# B&R Automation Studio project perfxxl (part 5)

#### motorman.c
```c
#ifdef _DEFAULT_INCLUDES
	#include <AsDefault.h>
#endif
/*
                             *******************
******************************* C SOURCE FILE *******************************
**                           *******************                           **
**                                                                         **
** project  : LS JET II                                                    **
** filename : MOTORMAN.C                                                   **
** version  : 1.11                                                         **
** date     : 08.11.2007                                                   **
**                                                                         **
*****************************************************************************
** Abstract                                                                **
** ========                                                                **
** Move motor manually                                                     **
**                                                                         **
**                                                                         **
** Copyright (c) 2006, Krause-Biagosch GmbH                                **
** All rights reserved.                                                    **
**                                                                         **
*****************************************************************************
VERSION HISTORY:
----------------
Version     : 1.00
Date        : 10.09.2002
Revised by  : Herbert Aden
Description : Original version.

Version     : 1.10
Date        : 07.11.2006
Revised by  : Herbert Aden
Description : -Code review, style improvement

Version     : 1.11
Date        : 08.11.2007
Revised by  : Herbert Aden
Description : - limits for checking movement are now always positive, and max>min
*/
#define _MOTORMAN_C_SRC

/****************************************************************************/
/**                                                                        **/
/**                           INCLUDE FILES                                **/
/**                                                                        **/
/****************************************************************************/
#include <string.h>
#include "asstring.h"
#include "glob_var.h"
#include "Motorfunc.h"

/****************************************************************************/
/**                                                                        **/
/**                       DEFINITIONS AND MACROS                           **/
/**                                                                        **/
/****************************************************************************/
/* NONE */

/****************************************************************************/
/**                                                                        **/
/**                      TYPEDEFS AND STRUCTURES                           **/
/**                                                                        **/
/****************************************************************************/
/* NONE */

/****************************************************************************/
/**                                                                        **/
/**                      PROTOTYPES OF LOCAL FUNCTIONS                     **/
/**                                                                        **/
/****************************************************************************/
/* NONE */

/****************************************************************************/
/**                                                                        **/
/**                      EXPORTED VARIABLES                                **/
/**                                                                        **/
/****************************************************************************/
/* NONE */

/****************************************************************************/
/**                                                                        **/
/**                           GLOBAL VARIABLES                             **/
/**                                                                        **/
/****************************************************************************/
_GLOBAL   UINT                ConveyorBeltOn;

/****************************************************************************/
/**                                                                        **/
/**                      TASK-LOCAL VARIABLES                              **/
/**                                                                        **/
/****************************************************************************/
_LOCAL    USINT               ManStep;
_LOCAL    USINT               MotorOnDisplay;
_LOCAL    USINT               ManPlus,ManMinus;

/****************************************************************************/
/**                                                                        **/
/**                    MODULE-LOCAL VARIABLES                              **/
/**                                                                        **/
/****************************************************************************/
static    DINT                tmpval;

/****************************************************************************/
/**                                                                        **/
/**                          EXPORTED FUNCTIONS                            **/
/**                                                                        **/
/****************************************************************************/
void MotorManual(void)
{
	MotorOnDisplay = gMotorOnDisplay;
	switch (ManStep)
	{
		case 0:
		{
			if(Motors[MotorOnDisplay].Error || MotorOnDisplay == 0)
				break;

/* don't start, if limit reached*/
			if ((MotorOnDisplay != CONVEYORBELT) && (MotorOnDisplay != ADJUSTER))
			{
				if( ( ManPlus &&
				      (labs(Motors[MotorOnDisplay].Position) > labs(Motors[MotorOnDisplay].Parameter.MaximumPosition))
				    )
				 ||
				    ( ManMinus &&
					 (labs(Motors[MotorOnDisplay].Position) < labs(Motors[MotorOnDisplay].Parameter.MinimumPosition))
				    )
				  )
				{
					break;
				}
			}

			if( ManPlus || ManMinus )
			{
				ManStep = 1;
				if( ManMinus )
					tmpval = (-1L) * labs(Motors[MotorOnDisplay].Parameter.ManSpeed);
				else
					tmpval = labs(Motors[MotorOnDisplay].Parameter.ManSpeed);
			}
			break;
		}
		case 1:
		{
			if (SendMotorCmd(MotorOnDisplay, CMD_SERIAL, FALSE, 0L ))
			{
				ManStep = 2;
			}
			break;
		}
		case 2:
		{
			if (SendMotorCmd(MotorOnDisplay, CMD_MOVE_AT, TRUE, tmpval ))
			{
				ManStep = 3;
			}
			break;
		}
		case 3:
		{
/*wait for key being released*/
/*V2.10 or limit reached*/
/*V2.13 build 22.06.2005 no limits for Motor 6 and 9 (Belt-motors)*/
			if ((MotorOnDisplay != CONVEYORBELT) && (MotorOnDisplay != ADJUSTER))
			{
				if( ( ManPlus &&
				      (labs(Motors[MotorOnDisplay].Position) > labs(Motors[MotorOnDisplay].Parameter.MaximumPosition))
				    )
				 ||
				    ( ManMinus &&
					 (labs(Motors[MotorOnDisplay].Position) < labs(Motors[MotorOnDisplay].Parameter.MinimumPosition))
				    )
				  )
				{
					ManStep = 4;
					break;
				}
			}

			if( ManPlus || ManMinus )
				break;
			else
				ManStep = 4;

			break;
		}
		case 4:
		{
			if (SendMotorCmd(MotorOnDisplay, CMD_STOP, FALSE, 0L) )
			{
				ManStep = 0;
				if(MotorOnDisplay == CONVEYORBELT)
					ConveyorBeltOn = FALSE;
			}
			break;
		}
	}
}
/****************************************************************************/
/**                                                                        **/
/**                                 EOF                                    **/
/**                                                                        **/
/****************************************************************************/
```

#### motortarget.c
```c
#ifdef _DEFAULT_INCLUDES
	#include <AsDefault.h>
#endif
/*
                             *******************
******************************* C SOURCE FILE *******************************
**                           *******************                           **
**                                                                         **
** project  : LS JET II                                                    **
** filename : MOTORTARGET.C                                                **
** version  : 1.11                                                         **
** date     : 12.10.2007                                                   **
**                                                                         **
*****************************************************************************
** Abstract                                                                **
** ========                                                                **
** Sequence for moving a motor to a certain position (manually)            **
**                                                                         **
**                                                                         **
** Copyright (c) 2006, Krause-Biagosch GmbH                                **
** All rights reserved.                                                    **
**                                                                         **
*****************************************************************************
VERSION HISTORY:
----------------
Version     : 1.00
Date        : 10.09.2002
Revised by  : Herbert Aden
Description : Original version.

Version     : 1.10
Date        : 07.11.2006
Revised by  : Herbert Aden
Description : -Code review, style improvement

Version     : 1.10
Date        : 12.10.2007
Revised by  : Herbert Aden
Description : MoveToAbsPosition has changed, so we must provide a pointer
              to an USINT variable that can hold the internal state of that fct.
*/
#define _MOTORTARGET_C_SRC

/****************************************************************************/
/**                                                                        **/
/**                           INCLUDE FILES                                **/
/**                                                                        **/
/****************************************************************************/
#include <string.h>
#include "asstring.h"
#include "glob_var.h"
#include "Motorfunc.h"

/****************************************************************************/
/**                                                                        **/
/**                       DEFINITIONS AND MACROS                           **/
/**                                                                        **/
/****************************************************************************/
/* NONE */

/****************************************************************************/
/**                                                                        **/
/**                      PROTOTYPES OF LOCAL FUNCTIONS                     **/
/**                                                                        **/
/****************************************************************************/
/* NONE */

/****************************************************************************/
/**                                                                        **/
/**                      EXPORTED VARIABLES                                **/
/**                                                                        **/
/****************************************************************************/
/* NONE */

/****************************************************************************/
/**                                                                        **/
/**                           GLOBAL VARIABLES                             **/
/**                                                                        **/
/****************************************************************************/
/* NONE */

/****************************************************************************/
/**                                                                        **/
/**                      TASK-LOCAL VARIABLES                              **/
/**                                                                        **/
/****************************************************************************/
_LOCAL USINT	TargetStep;
_LOCAL USINT	MotorOnDisplay;
_LOCAL USINT	TargetStart;
_LOCAL DINT	TargetPosition;

/****************************************************************************/
/**                                                                        **/
/**                    MODULE-LOCAL VARIABLES                              **/
/**                                                                        **/
/****************************************************************************/
static    USINT               MotStep;       /* holds current step of fct MoveToAbsPosition */

/****************************************************************************/
/**                                                                        **/
/**                          EXPORTED FUNCTIONS                            **/
/**                                                                        **/
/****************************************************************************/
void MotorTarget(void)
{
	switch (TargetStep)
	{
		case 0:
		{
			if(		(Motors[MotorOnDisplay].Error == TRUE)
			    ||  (Motors[MotorOnDisplay].ReferenceOk == FALSE)
				||	(MotorOnDisplay == 0) )
				break;

/*check limit positions*/
			if ((MotorOnDisplay != CONVEYORBELT) && (MotorOnDisplay != ADJUSTER))
			{
				if(		(labs(TargetPosition) > labs(Motors[MotorOnDisplay].Parameter.MaximumPosition) )
					||	(labs(TargetPosition) < labs(Motors[MotorOnDisplay].Parameter.MinimumPosition)) )
					break;
			}

			if( TargetStart)
			{
				TargetStep = 1;
				TargetStart = FALSE;
			}
			break;
		}
		case 1:
		{
/*wait, till no other sending active*/
			if( MoveToAbsPosition(MotorOnDisplay,
			                      TargetPosition,
			                      Motors[MotorOnDisplay].Parameter.ManSpeed,
			                      &MotStep) )
			{
				TargetStep = 4;
			}
			break;
		}
		case 4:
		{
/*set maximum speed*/
			if( SendMotorCmd(MotorOnDisplay,
			                 CMD_SPEED,
			                 TRUE,
			                 Motors[MotorOnDisplay].Parameter.MaximumSpeed) )
			{
				TargetStep = 0;
			}
			break;
		}
	}
/*always reset the start command unconditionally*/
	TargetStart = FALSE;

}
/****************************************************************************/
/**                                                                        **/
/**                                 EOF                                    **/
/**                                                                        **/
/****************************************************************************/
```

#### motorstop.c
```c
#ifdef _DEFAULT_INCLUDES
	#include <AsDefault.h>
#endif
/****************************************************************************/
/*	Stoppen aller Motoren (quasi NOTAUS)*/
/*																			*/
/*																			*/
/*	Versionsgeschichte:														*/
/*  Version		Datum		Änderung								von		*/
/*	1.0			30.06.03	erste Implementation					HA		*/
/*																			*/
/*																			*/
/****************************************************************************/
#include "glob_var.h"
#include "in_out.h"
#include "asstring.h"
#include <string.h>
#include "motorfunc.h"

#define BROADCAST 127

_LOCAL 	USINT	StopStep;
_LOCAL F_TRIGtyp F_DoorSensor;

_GLOBAL	BOOL	StopMotors;
_GLOBAL	BOOL	ReferenceStart;

USINT	 		tmp[20];
USINT	i;

void MotorStop(void)
{

	AlarmBitField[27] = !DoorsOK;

	F_DoorSensor.CLK = DoorsOK;
/*CoverLockOn ist das Zeichen dafür, dass ein Ablauf aktiv sein muss, nur dann muss alles gestoppt werden!*/
	F_TRIG(&F_DoorSensor);

	if( F_DoorSensor.Q && Out_CoverLockOn ) StopMotors = 1;

	switch (StopStep)
	{
		case 0:
		{
			i = 0;
			if( StopMotors )
				StopStep = 2;
			break;
		}

		case 2:
		{
/*stop all sequences*/
			START = 0;
			AUTO = 0;
			PaperRemoveStart = 0;
			PaperRemoveStart = 0;
			PlateTakingStart = 0;
			AdjustStart = 0;
			DeloadStart = 0;
			ExposeStart = 0;
			CloseTrolleyStart = 0;
			OpenTrolleyStart = 0;
			ReferenceStart = 0;

/*release cover lock*/
			Out_CoverLockOn = 0;

/*stop LUST Controller*/
			FU.cmd_Start = 0;
			FU.cmd_Auto = 0;

			for(i=0;i<MotorsConnected;i++)
			{
				Motors[i].ReferenceOk = 0;
				Motors[i].StartRef = 0;
				Motors[i].ReferenceStep = 0;
			}

			StopStep = 5;
			break;
		}

		case 5:
		{
/*wait, till no other sending active*/
/*send V0 to all motors at once (BROADCAST)*/
			if (SendMotorCmd(BROADCAST,"V0",0,0))
				StopStep = 10;
			break;
		}
/*reset reference ok flags*/
		case 10:
		{
			StopStep = 15;
			break;
		}

		case 15:
		{
				if(wBildAktuell != 41 )
					OrgBild = wBildAktuell;
				wBildNeu = 41;
				AbfrageOK = 0;
				AbfrageCancel = 0;
				IgnoreButtons = 0;
				OK_CancelButtonInv = 1;
				OK_ButtonInv = 0;
				AbfrageText1 = 43;
				AbfrageText2 = 45;
				AbfrageText3 = 46;
				AbfrageIcon = CAUTION;
				StopStep = 20;
			break;
		}
		case 20:
		{
			if(AbfrageOK)
			{
				AbfrageOK = 0;
				StopStep = 0;
				StopMotors = 0;
			}
			break;
		}
	}
}
```

- motorfunc.h (reference to Logical/GlobalIncludes/motorfunc.h)

- glob_var.h (reference to Logical/GlobalIncludes/glob_var.h)

#### auxfunc.c
```c
#ifdef _DEFAULT_INCLUDES
	#include <AsDefault.h>
#endif
/*
                             *******************
******************************* C SOURCE FILE *******************************
**                           *******************                           **
**                                                                         **
** project  : LS JET II                                                    **
** filename : AUXFUNC.C                                                    **
** version  : 1.00                                                         **
** date     : 27.10.2006                                                   **
**                                                                         **
*****************************************************************************
** Abstract                                                                **
** ========                                                                **
** Implementation of function for common use, e.g. showing an error        **
** message                                                                 **
**                                                                         **
** Copyright (c) 2006, Krause-Biagosch GmbH                                **
** All rights reserved.                                                    **
**                                                                         **
*****************************************************************************
VERSION HISTORY:
----------------
Version     : 1.00
Date        : 27.10.2006
Revised by  : Herbert Aden
Description : Original version.
*/
#define _AUXFUNC_C_SRC

/****************************************************************************/
/**                                                                        **/
/**                           INCLUDE FILES                                **/
/**                                                                        **/
/****************************************************************************/
#include "glob_var.h"
#include "in_out.h"
#include "egmglob_var.h"
#include "asstring.h"
#include <string.h>

#include "auxfunc.h"

/****************************************************************************/
/**                                                                        **/
/**                       DEFINITIONS AND MACROS                           **/
/**                                                                        **/
/****************************************************************************/
/* NONE */

/****************************************************************************/
/**                                                                        **/
/**                      EXPORTED VARIABLES                                **/
/**                                                                        **/
/****************************************************************************/
/*@checked@*/

/****************************************************************************/
/**                                                                        **/
/**                           GLOBAL VARIABLES                             **/
/**                                                                        **/
/****************************************************************************/
_GLOBAL	UINT	EmptyReturnPic;

/****************************************************************************/
/**                                                                        **/
/**                          EXPORTED FUNCTIONS                            **/
/**                                                                        **/
/****************************************************************************/
void ShowMessage(const int T1,const int T2,const int T3,
                 const int Icon, const int Button, const BOOL pIgnoreButtons)
{
	switch (Button)
	{
		case NONE:
		{
			OK_CancelButtonInv = TRUE;
			OK_ButtonInv = TRUE;
			break;
		}
		case OKONLY:
		{
			OK_CancelButtonInv = TRUE;
			OK_ButtonInv = FALSE;
			break;
		}
		case OKCANCEL:
		{
			OK_CancelButtonInv = FALSE;
			OK_ButtonInv = TRUE;
			break;
		}
		default:
		{
			break;
		}
	}
	AbfrageIcon = Icon;
	AbfrageText1 = T1;
	AbfrageText2 = T2;
	AbfrageText3 = T3;
	IgnoreButtons = pIgnoreButtons;
	if(wBildAktuell != MESSAGEPIC )
	{
		if(wBildAktuell == EMPTYPIC)
		{
			if(EmptyReturnPic != MESSAGEPIC)
				OrgBild = EmptyReturnPic;
		}
		else
			OrgBild = wBildAktuell;
	}
	wBildNeu = MESSAGEPIC;
	AbfrageOK = 0;
	AbfrageCancel = 0;
}

void SwitchFeederVacuum(USINT PlateType, USINT Config, BOOL fct)
{
	switch (Config)
	{
		case LEFT:
		{
			Out_FeederVacuumOn[0] = fct;
			Out_FeederVacuumOn[2] = fct;
			break;
		}
		case RIGHT:
		{
			Out_FeederVacuumOn[1] = fct;
			Out_FeederVacuumOn[3] = fct;
			break;
		}
		case BOTH:
		{
			Out_FeederVacuumOn[0] = fct;
			Out_FeederVacuumOn[1] = fct;
			Out_FeederVacuumOn[2] = fct;
			Out_FeederVacuumOn[3] = fct;
			break;
		}
		case PANORAMA:
		{
			switch (PlateType)
			{
				case 1:
				{
					Out_FeederVacuumOn[0] = fct;
					Out_FeederVacuumOn[1] = fct;
					break;
				}
				case 2:
				{
					Out_FeederVacuumOn[0] = fct;
					Out_FeederVacuumOn[1] = fct;
					Out_FeederVacuumOn[2] = fct;
					Out_FeederVacuumOn[3] = fct;
					break;
				}
				default:
				{
					Out_FeederVacuumOn[1] = fct;
					Out_FeederVacuumOn[3] = fct;
					break;
				}
			}
/*
			Out_FeederVacuumOn[0] = fct;
			Out_FeederVacuumOn[1] = fct;
			Out_FeederVacuumOn[2] = fct;
			Out_FeederVacuumOn[3] = fct;
*/
			break;
		}
		case BROADSHEET:
		{
			Out_FeederVacuumOn[0] = fct;
			Out_FeederVacuumOn[1] = fct;
			Out_FeederVacuumOn[4] = fct;
			break;
		}
		case ALL:
		{
			Out_FeederVacuumOn[0] = fct;
			Out_FeederVacuumOn[1] = fct;
			Out_FeederVacuumOn[2] = fct;
			Out_FeederVacuumOn[3] = fct;
			Out_FeederVacuumOn[4] = fct;
			break;
		}
	}
}

void SwitchAdjustVacuum(USINT PlateType, USINT Config, BOOL fct)
{
	switch (Config)
	{
		case LEFT:
		{
			Out_AdjustSuckerVacuumOn[0] = fct;
			break;
		}
		case RIGHT:
		{
			Out_AdjustSuckerVacuumOn[1] = fct;
			break;
		}
		case BOTH:
		{
			Out_AdjustSuckerVacuumOn[0] = fct;
			Out_AdjustSuckerVacuumOn[1] = fct;
			break;
		}
		case PANORAMA:
		{
			Out_AdjustSuckerVacuumOn[0] = fct;
			Out_AdjustSuckerVacuumOn[1] = fct;
			break;
		}
		case BROADSHEET:
		{
			Out_AdjustSuckerVacuumOn[2] = fct;
			break;
		}
		case ALL:
		{
			Out_AdjustSuckerVacuumOn[0] = fct;
			Out_AdjustSuckerVacuumOn[1] = fct;
			Out_AdjustSuckerVacuumOn[2] = fct;
			break;
		}
	}
}

void SwitchAdjustTableVacuum(USINT PlateType, USINT Config, BOOL fct)
{
	switch (Config)
	{
		case LEFT:
		{
			AdjustVacuumOn[0] = fct;
			AdjustVacuumOn[2] = fct;
			break;
		}
		case RIGHT:
		{
			AdjustVacuumOn[1] = fct;
			AdjustVacuumOn[2] = fct;
			break;
		}
		case BOTH:
		{
			AdjustVacuumOn[0] = fct;
			AdjustVacuumOn[1] = fct;
			AdjustVacuumOn[2] = fct;
			break;
		}
		case PANORAMA:
		{
			switch (PlateType)
			{
				case 1:
				{
					AdjustVacuumOn[0] = fct;
					break;
				}
				case 2:
				{
					AdjustVacuumOn[0] = fct;
					AdjustVacuumOn[1] = fct;
					break;
				}
			}
/*
			AdjustVacuumOn[0] = fct;
			AdjustVacuumOn[1] = fct;
			AdjustVacuumOn[2] = fct;
*/
			break;
		}
		case BROADSHEET:
		{
			AdjustVacuumOn[2] = fct;
			break;
		}
		case ALL:
		{
			AdjustVacuumOn[0] = fct;
			AdjustVacuumOn[1] = fct;
			AdjustVacuumOn[2] = fct;
			break;
		}
	}
}

/****************************************************************************/
/* Hilfsfunktion: Papiersensoren prüfen */
/* PlateSet                     */
/* LEFT, RIGHT, BOTH/PANO, BROADSHEET */
/****************************************************************************/
BOOL CheckForPaper(USINT Config)
{
	BOOL PaperDetected = FALSE;
	switch (Config)
	{
		case LEFT:
		{
			PaperDetected = In_PaperSensor[0];
			break;
		}
		case RIGHT:
		{
			PaperDetected = In_PaperSensor[1];
			break;
		}
		case BOTH:
		{
			PaperDetected = In_PaperSensor[0] || In_PaperSensor[1];
			break;
		}
		case PANORAMA:
		{
			PaperDetected = In_PaperSensor[0] || In_PaperSensor[1];
			break;
		}
		case BROADSHEET:
		{
			PaperDetected = In_PaperSensor[0] || In_PaperSensor[1];
			break;
		}
	}

	if(!GlobalParameter.PaperRemoveEnabled || PlateTransportSim)
		PaperDetected = FALSE;

	return PaperDetected;

}

/****************************************************************************/
/* Hilfsfunktion: Vakuum prüfen */
/* PlateSet                     */
/* LEFT, RIGHT, BOTH/PANO, BROADSHEET */
/****************************************************************************/
BOOL CheckFeederVacuum(USINT PlateType, USINT Config)
{
	BOOL VacuumOK = FALSE;

	switch (Config)
	{
		case LEFT:
		{
			VacuumOK = In_FeederVacuumOK[0] && In_FeederVacuumOK[2];
			break;
		}
		case RIGHT:
		{
			VacuumOK = In_FeederVacuumOK[1] && In_FeederVacuumOK[3];
			break;
		}
		case BOTH:
		{
			VacuumOK = In_FeederVacuumOK[0] && In_FeederVacuumOK[1]
			        && In_FeederVacuumOK[2] && In_FeederVacuumOK[3];
			break;
		}
		case PANORAMA:
		{
			switch (PlateType)
			{
				case 1:
				{
					VacuumOK = In_FeederVacuumOK[0] && In_FeederVacuumOK[1];
					break;
				}
				case 2:
				{
					VacuumOK = In_FeederVacuumOK[0] && In_FeederVacuumOK[1]
								&& In_FeederVacuumOK[2] && In_FeederVacuumOK[3];
					break;
				}
				default:
				{
					VacuumOK = In_FeederVacuumOK[1] && In_FeederVacuumOK[3];
					break;
				}
			}
/*
			VacuumOK = In_FeederVacuumOK[0] && In_FeederVacuumOK[1]
			        && In_FeederVacuumOK[2] && In_FeederVacuumOK[3];
*/
			break;
		}
		case BROADSHEET:
		{
			VacuumOK = In_FeederVacuumOK[0]
			        && In_FeederVacuumOK[1]
			        && In_FeederVacuumOK[4];
			break;
		}
	}

	if(PlateTransportSim)
		VacuumOK = TRUE;
	return VacuumOK;
}

/****************************************************************************/
/* Hilfsfunktion: Vakuum prüfen */
/* PlateSet                     */
/* LEFT, RIGHT, BOTH/PANO, BROADSHEET */
/****************************************************************************/
BOOL CheckAdjustVacuum(USINT PlateType, USINT Config)
{
	BOOL VacuumOK = FALSE;
	switch (Config)
	{
		case LEFT:
		{
			VacuumOK = In_AdjustVacuumOK[0];
			break;
		}
		case RIGHT:
		{
			VacuumOK = In_AdjustVacuumOK[1];
			break;
		}
		case BOTH:
		{
			VacuumOK = In_AdjustVacuumOK[0] && In_AdjustVacuumOK[1];
			break;
		}
		case PANORAMA:
		{
			VacuumOK = In_AdjustVacuumOK[0];
			break;
		}
		case BROADSHEET:
		{
			VacuumOK = In_AdjustVacuumOK[0];
			break;
		}
	}

	if(PlateTransportSim)
		VacuumOK = TRUE;

	return VacuumOK;

}

void MoveAdjustSucker(USINT Config, USINT fct)
{
	switch (Config)
	{
		case LEFT:
		{
			Out_AdjustSuckerActive[0] = fct;
			break;
		}
		case RIGHT:
		{
			Out_AdjustSuckerActive[1] = fct;
			Out_AdjustSuckerActive[2] = fct;
			break;
		}
		case BOTH:
		{
			Out_AdjustSuckerActive[0] = fct;
			Out_AdjustSuckerActive[1] = fct;
			Out_AdjustSuckerActive[2] = fct;
			break;
		}
		case PANORAMA:
		{
			Out_AdjustSuckerActive[0] = fct;
			Out_AdjustSuckerActive[1] = fct;
			Out_AdjustSuckerActive[2] = fct;
			break;
		}
		case BROADSHEET:
		{
			Out_AdjustSuckerActive[2] = fct;
			break;
		}
		case ALL:
		{
			Out_AdjustSuckerActive[0] = fct;
			Out_AdjustSuckerActive[1] = fct;
			Out_AdjustSuckerActive[2] = fct;
			break;
		}
	}
}

BOOL AdjustOK(USINT Config)
{
	BOOL retval = FALSE;
	switch (Config)
	{
		case LEFT:
		{
			retval = In_PlateAdjusted[0];
			break;
		}
		case RIGHT:
		{
			retval = In_PlateAdjusted[1];
			break;
		}
		case BOTH:
		{
			retval = In_PlateAdjusted[0] && In_PlateAdjusted[0];
			break;
		}
		case PANORAMA:
		{
			retval = In_PlateAdjusted[0];
			break;
		}
		case BROADSHEET:
		{
			retval = In_PlateAdjusted[0];
			break;
		}
	}
	if(PlateTransportSim || AdjusterParameter.AdjustSim)
		retval = TRUE;

	return retval;
}

BOOL AdjPins(USINT Config,USINT *Step, TON_10ms_typ *Timer)
{
	BOOL retval = FALSE;

	if(Config == LEFT)
		return TRUE;
/* Panorama plate or down command: all pins down*/
	if( (Config == PANORAMA)
	 || (Config == PINS_DOWN)
	  )
	{
		switch (*Step)
		{
			case 0:
			{
/* schon unten? -> nichts zu tun, weiter*/
				if(  Out_AdjustPinsDown
				 && !Out_AdjustPins4and6Up
				 && !Out_AdjustPin3Up)
				{
					*Step = 0;
					Timer->IN = FALSE;
					retval = TRUE;
					break;
				}
/* erstmal senken ansteuern */
				if(Timer->Q && Out_AdjustPinsDown)
				{
					Timer->IN = FALSE;
					*Step = 10;
					break;
				}
				Timer->IN = TRUE;
				Timer->PT = 10;
				Out_AdjustPinsDown = ON;
				break;
			}
			case 10:
			{
				if(Timer->Q && !Out_AdjustPins4and6Up && !Out_AdjustPin3Up)
				{
					Timer->IN = FALSE;
					*Step = 20;
					break;
				}
				Timer->IN = TRUE;
				Timer->PT = AdjusterParameter.PinsDownTime;
				Out_AdjustPins4and6Up = OFF;
				Out_AdjustPin3Up = OFF;
				break;
			}
			case 20:
			{
				*Step = 0;
				Timer->IN = FALSE;
				retval = TRUE;
				break;
			}
		}
	}
	else
	{
		switch (*Step)
		{
			case 0:
			{
/* pin config fits plate config: nothing to do, just end*/
				if(  ( (Config == BROADSHEET)
					 && !Out_AdjustPins4and6Up
					 && Out_AdjustPin3Up
					 && !Out_AdjustPinsDown
					 )
				 ||  (((Config == BOTH) || (Config == RIGHT))
					 && Out_AdjustPins4and6Up
					 && Out_AdjustPin3Up
					 && !Out_AdjustPinsDown
				     )
				  )
				{
					retval = TRUE;
					break;
				}
/* Cross: only pin 3 may be up*/
				if( (Config == BROADSHEET)
				 &&  Out_AdjustPins4and6Up
				  )
				{
					*Step = 2;
					Timer->IN = FALSE;
					break;
				}
/* both or right: pins 3,4 and 6 must be up */
				Out_AdjustPinsDown = ON;
				*Step = 10;
				Timer->IN = FALSE;

				break;
			}
/**************************/
/* pins 4 and 6 down for cross format*/
			case 2:
			{
				if(Timer->Q && Out_AdjustPinsDown)
				{
					Timer->IN = FALSE;
					*Step = 4;
					break;
				}
				Out_AdjustPinsDown = ON;
				Timer->IN = TRUE;
				Timer->PT = 10;
				break;
			}
			case 4:
			{
				if(Timer->Q && !Out_AdjustPins4and6Up)
				{
					Timer->IN = FALSE;
					*Step = 10;
					break;
				}
				Out_AdjustPins4and6Up = OFF;
				Timer->IN = TRUE;
				Timer->PT = AdjusterParameter.PinsDownTime;
				break;
			}
/**************************/
			case 10:
			{
				if(Timer->Q && Out_AdjustPin3Up)
				{
					*Step = 20;
					Timer->IN = FALSE;
					break;
				}
				if( (Config == RIGHT)
				 || (Config == BOTH)
				  )
					Out_AdjustPins4and6Up = ON;
	/* pin 3 must always be up */
				Out_AdjustPin3Up = ON;
				Timer->IN = TRUE;
				Timer->PT = 10;
				break;
			}

			case 20:
			{
				if(Timer->Q && !Out_AdjustPinsDown)
				{
					Timer->IN = FALSE;
					*Step = 0;
					retval = TRUE;
					break;
				}
				Out_AdjustPinsDown = OFF;
				Timer->IN = TRUE;
				Timer->PT = AdjusterParameter.PinsDownTime;
				break;
			}
		}
	}
	return retval;
}

void ClearStation(PlateInSystem_Type *Station)
{
	Station->present = FALSE;
/*	Station->PlateConfig = NOPLATE;*/
	Station->PlateType = 0;
	Station->NextPlateType = 0;
	strcpy(Station->FileName,"");
	Station->ErrorCode = 0;
	strcpy(Station->ID,"");
	Station->Status = 0;
}

/****************************************************************************/
/**                                                                        **/
/**                                 EOF                                    **/
/**                                                                        **/
/****************************************************************************/
```

- auxfunc.h (reference to Logical/GlobalIncludes/auxfunc.h)

### Program Logical/Exposer/Hardware/lust_cdd (ANSIC, version 1.10.0) - LUST CDD3000 Treiber

#### lust_cdd.c
```c
#ifdef _DEFAULT_INCLUDES
	#include <AsDefault.h>
#endif
/****************************************************************************/
/*	Treiberprogramm für LUST FU CDD3000 über CAN		 					*/
/*																			*/
/*																			*/
/*	Versionsgeschichte:														*/
/*  Version		Datum		Änderung								von		*/
/*	1.10		13.08.02	zyklische Übertragung des Steuerwortes	HA		*/
/*	1.00		06.08.02	erste Implementation					HA		*/
/*																			*/
/*																			*/
/****************************************************************************/
#include <string.h>					/*	Definitionen für Stringfunktionen	*/

#include "standard.h"
#include "sys_lib.h"

#include "bit_func.h"				/*	Macros für die Bitbearbeitung		*/
#include "glob_var.h"

/****************************************************************************/
/*		DEFINES																*/
/****************************************************************************/
#define STANDARD_PARAM_ENQ 5
#define STANDARD_PARAM_SEL 2
#define FELD_PARAM_ENQ 13
#define FELD_PARAM_SEL 12

#define WAITCYCLES		15
#define	TIMEOUT			50

/****************************************************************************/
/*		Variablendeklaration												*/
/****************************************************************************/
_GLOBAL	plcbit			CAN_ok;

/* Hilfsvariable für Watch */
_GLOBAL BOOL FU_INIT_RDY;

/* Struktur als Schnittstelle zur Applikation */
_GLOBAL	FU_Typ 			FU;

/* Struktur für zu schreibende/lesende Parameter */
_GLOBAL	FU_Para_Typ		FU_Param;

/* Struktur für die eigentlichen Telegrammdaten								*/
_GLOBAL	CAN_OBJEKT_FUtyp	Can_FU;

_LOCAL unsigned short i;
DINT* tmpPtr;
_GLOBAL BOOL MirroredMachine;
_LOCAL REAL ParkSpeed_Old;
extern REAL 	speed_old,StartPosition_old,PEGStartPosition_old,EndPosition_old,
		PEGEndPosition_old;

/****************************************************************************/
/*		Prototypen															*/
/****************************************************************************/
extern void ReferenzFahrt(void);
extern void resetFUData(void);
extern void ParkPosition(void);
extern void ZielPosition(void);
extern void Belichtung(void);

/****************************************************************************/
/*		Initialisierungs-UP													*/
/*   																		*/
/****************************************************************************/
_INIT void lust_cdd_init(void)
{
	FU_INIT_RDY = FALSE;
	FU.Status = 0;
	FU.ParaStep = 0;
	FU_Param.Error = 0;
	FU_Param.Ready = 0;
	strcpy(&FU.DrvError[0],"Init...");
	resetFUData();
	FU.CANError = TRUE;
	speed_old = 0.0;
	StartPosition_old = 0.0;
	PEGStartPosition_old = 0.0;
	EndPosition_old = 0.0;
	PEGEndPosition_old = 0.0;
	ParkSpeed_Old = 0.0;
}

/****************************************************************************/
/*		zyklischer Teil      												*/
/****************************************************************************/
_CYCLIC void lust_cdd_cyclic(void)
{
	int j;
/* Funktionen aufrufen*/
	ReferenzFahrt();
	ParkPosition();
	ZielPosition();
	Belichtung();

/* CAN nicht ok? dann ende */
	if (CAN_ok != 1)				/* Fehler aus 'can_comm' Task */
	{
		strcpy(&FU.DrvError[0],"CANERROR");
		resetFUData();
		FU.CANError = TRUE;
		return;
	}
/* CAN ist ok, also weiter*/

/* FU meldet sich nach dem Einschalten auf BAsis ID $607 */
	if (Can_FU.InitResEv == 1)
	{
			FU_INIT_RDY = 1;

	/* FU init quittieren, Antwort mit $dd */
			Can_FU.InitResEv = 0;
			Can_FU.InitReq[0] = 1;
			Can_FU.InitReqEv = 1;
/* Variablen initialisieren */
			FU.SetPara = 0;
			FU.GetPara = 0;
			FU.IndexPara = 0;
			FU.IdxIntern = 0;
			FU.timeoutCounter = 0;
			resetFUData();
			strcpy(&FU.DrvError[0],"INIT OK");
			FU.CANError = FALSE;
	}

/********************************************************************/
/* 																	*/
/* FU meldet seinen Status nach dem Initialisieren auf Basis $371   */
/* dieses Telegramm kommt zyklisch vom Antrieb, deshalb hier		*/
/* über Timeout Erkennung, ob Antrieb noch am Bus					*/
/* 																	*/
/********************************************************************/

	if (Can_FU.StatResEv == 1)
	{
			FU.CANError = FALSE;
			Can_FU.StatResEv = 0;
			FU.Status = Can_FU.StatRes[0];
/* Statusinformationen in Einzelbits eintragen */
		/* Byte 0 */
			FU.Error 			= BIT_TST(Can_FU.StatRes[0],0);
			FU.CANStatus		= BIT_TST(Can_FU.StatRes[0],1);
			FU.SollwertErreicht	= BIT_TST(Can_FU.StatRes[0],2);
			FU.Activ 			= BIT_TST(Can_FU.StatRes[0],4);
			FU.Rot0 			= BIT_TST(Can_FU.StatRes[0],5);
			FU.CReady 			= BIT_TST(Can_FU.StatRes[0],7);
		/* Byte 1*/
			FU.ENPO 			= BIT_TST(Can_FU.StatRes[1],0);
			FU.OSD00 			= BIT_TST(Can_FU.StatRes[1],1);
			FU.OSD01 			= BIT_TST(Can_FU.StatRes[1],2);
		/* Byte 2 */
			FU.RefOk 			= BIT_TST(Can_FU.StatRes[2],0);
			FU.Auto 			= BIT_TST(Can_FU.StatRes[2],1);
			FU.Ablauf 			= BIT_TST(Can_FU.StatRes[2],2);
			for (i=0;i<8;i++)
			{
				FU.ZustandsMerker[i] =  BIT_TST(Can_FU.StatRes[3],i);
			}
		/* aktuelle Pos aus bytes 4..7 */
			tmpPtr =(UDINT*) &Can_FU.StatRes[4];
			FU.aktuellePosition = *tmpPtr;
			FU.aktuellePosition_mm = ((float) FU.aktuellePosition)/X_Param.InkrementeProMm;

			FU.timeoutCounter = 0;
			strcpy(&FU.DrvError[0],"STAT OK");

	}
/* timeout überwachung */
	else
	{
			FU.timeoutCounter ++;
			if (FU.timeoutCounter >= TIMEOUT)
			{
				strcpy(&FU.DrvError[0],"Timeout");
				FU.timeoutCounter = 0;
				CAN_ok = 0;
				resetFUData();
				FU.CANError = TRUE;
			}

	}

/********************************************************************/
/* 																	*/
/* Steuerwort senden zyklisch										*/
/* 																	*/
/********************************************************************/

/* kein ENPO -> steuerdaten alle 0*/
	if (!FU.ENPO)
	{
		FU.IdxIntern = 0;
		for (i=0;i<8;i++)
			Can_FU.SteuReq[i] = 0;
/*HA 18.05.2005 V2.11 reset start commands if no ENPO*/
		FU.cmd_Start = 0;
		FU.cmd_Auto = 0;
	}

/********************************************************************/
/* falls Fehler: quittieren  */
	if (FU.Error)
	{
/* erst Fehler Quittierung AUS */
		if(FU.IdxIntern <= WAITCYCLES)
		{
			FU.IdxIntern++;
			if(FU.IdxIntern == WAITCYCLES)
			{
				Can_FU.SteuReq[0] = 0 ; /*  */
				FU.IdxIntern = 300;
				FU.cmd_Start = 0;
			}
		}
		else
/* dann Fehler Quittierung EIN (Flanke erzeugen)*/
		{
			if(FU.IdxIntern <= 300+WAITCYCLES)
			{
				FU.IdxIntern++;
				if(FU.IdxIntern == 300+WAITCYCLES)
				{
					Can_FU.SteuReq[0] = 128; /*  */
					FU.IdxIntern = 0;
				}
			}
		} /* else */
	} /*if (FU.Error)*/

/********************************************************************/
/* Befehl aus App: Regelung freigeben*/
	if(FU.cmd_Start)
	{
	/* Regelung nicht aktiv */
		if (!FU.Activ)
		{
	/* erst Regelung gezielt AUS schalten*/
			if(FU.IdxIntern <= WAITCYCLES)
			{
				FU.IdxIntern++;
				if(FU.IdxIntern == WAITCYCLES)
				{
					Can_FU.SteuReq[0] = BIT_CLR(Can_FU.SteuReq[0],0); /* Regelung AUS */
					Can_FU.SteuReq[2] = BIT_CLR(Can_FU.SteuReq[2],0); /* Auto AUS*/
					Can_FU.SteuReq[2] = BIT_CLR(Can_FU.SteuReq[2],1); /* Ablauf AUS*/
					FU.IdxIntern = 300;
				}
			} /*if(FU.IdxIntern <= 8)*/
	/* dann Regelung gezielt wieder EIN schalten*/
			else
			{
				FU.IdxIntern++;
				if(FU.IdxIntern == 300+WAITCYCLES)
				{
					Can_FU.SteuReq[0] = BIT_SET(Can_FU.SteuReq[0],0); /* Regelung EIN */
					Can_FU.SteuReq[2] = BIT_CLR(Can_FU.SteuReq[2],0); /* Auto AUS*/
					Can_FU.SteuReq[2] = BIT_CLR(Can_FU.SteuReq[2],1); /* Ablauf AUS*/
					FU.IdxIntern = 0;
				}
			} /*else*/
		} /*if (!FU.Activ)*/
	} /*if(FU.cmd_Start)*/
	else
/* Befehl aus App: Reglerfreigabe AUS */
	{
	/* Regelung aktiv */
		if (FU.Activ)
		{
	/* Regelung gezielt AUS schalten*/
			FU.IdxIntern++;
			if(FU.IdxIntern == WAITCYCLES)
			{
				Can_FU.SteuReq[0] = BIT_CLR(Can_FU.SteuReq[0],0); /* Regelung AUS */
				Can_FU.SteuReq[2] = BIT_CLR(Can_FU.SteuReq[2],0); /* Auto AUS*/
				Can_FU.SteuReq[2] = BIT_CLR(Can_FU.SteuReq[2],1); /* Ablauf AUS*/
				FU.IdxIntern = 0;
			} /*if(FU.IdxIntern == 8)*/
		}/* if (FU.Activ)*/
	} /*else*/

/********************************************************************/
/* nur wenn aus App AUTO Befehl kommt... */
	if (FU.cmd_Auto && !FU.state_tipp_plus && !FU.state_tipp_minus)
	{
/*nach kurzer Zeit Automatik EIN schalten*/
		if (FU.Activ && !FU.Auto)
		{
			FU.IdxIntern++;
			if(FU.IdxIntern == WAITCYCLES)
			{
				Can_FU.SteuReq[2] = BIT_SET(Can_FU.SteuReq[2],0); /*Auto EIN*/
				Can_FU.SteuReq[2] = BIT_CLR(Can_FU.SteuReq[2],1); /*Ablauf AUS*/

				FU.IdxIntern = 0;
				FU.cmd_tipp_schnell = 0;
			}
		}

/*nach kurzer Zeit Ablaufprogramm Start EIN schalten*/
		if (FU.Activ && FU.Auto && !FU.Ablauf)
		{
			FU.IdxIntern++;
			if(FU.IdxIntern == WAITCYCLES)
			{
				Can_FU.SteuReq[2] = BIT_SET(Can_FU.SteuReq[2],1); /*Ablauf EIN*/
				FU.IdxIntern = 0;
			}
		}
	} /* if cmd_Auto */
/* sonst Handbetrieb */
	else
/*nach kurzer Zeit Automatik AUS schalten*/
	{
		if (FU.Auto && !FU.state_tipp_plus && !FU.state_tipp_minus)
		{
			FU.IdxIntern++;
			if(FU.IdxIntern == WAITCYCLES)
			{
				Can_FU.SteuReq[2] = BIT_CLR(Can_FU.SteuReq[2],0); /*Auto AUS*/
				Can_FU.SteuReq[2] = BIT_CLR(Can_FU.SteuReq[2],1); /*Ablauf AUS*/
				Can_FU.SteuReq[2] = BIT_CLR(Can_FU.SteuReq[2],6); /*TIPP+*/
				Can_FU.SteuReq[2] = BIT_CLR(Can_FU.SteuReq[2],7); /*TIPP-*/
				FU.cmd_tipp_plus = 0;
				FU.cmd_tipp_minus = 0;
				FU.state_tipp_plus = 0;
				FU.state_tipp_minus = 0;
				FU.state_tipp_schnell = 0;

				FU.IdxIntern = 0;
			}
		}
		else /* wenn Auto AUS ist */
		{
/*  TIPP Betrieb auswerten */

/****** PLUS ****/
/* Kommando TIPP + gekommen: einmal TIPP+ Bit setzen */
			if (FU.cmd_tipp_plus && !FU.state_tipp_plus )
			{
				if (MirroredMachine)
					Can_FU.SteuReq[2] = BIT_SET(Can_FU.SteuReq[2],7); /*TIPP-*/
				else
					Can_FU.SteuReq[2] = BIT_SET(Can_FU.SteuReq[2],6); /*TIPP+*/
				FU.state_tipp_plus = 1;
				FU.IdxIntern = 0;
			}

/****** MINUS ****/
/* Kommando TIPP- gekommen: einmal TIPP- Bit setzen */
			if (FU.cmd_tipp_minus && !FU.state_tipp_minus )
			{
				if (MirroredMachine)
					Can_FU.SteuReq[2] = BIT_SET(Can_FU.SteuReq[2],6); /*TIPP+*/
				else
					Can_FU.SteuReq[2] = BIT_SET(Can_FU.SteuReq[2],7); /*TIPP-*/
				FU.state_tipp_minus = 1;
				FU.IdxIntern = 0;
			}

/* Schnell: zusätzlich das andere Bit setzen */
			if (FU.state_tipp_plus && FU.cmd_tipp_schnell && !FU.state_tipp_schnell)
			{
				FU.IdxIntern ++;
				if(	FU.IdxIntern == WAITCYCLES )
				{
					if (MirroredMachine)
						Can_FU.SteuReq[2] = BIT_SET(Can_FU.SteuReq[2],6); /*TIPP-*/
					else
						Can_FU.SteuReq[2] = BIT_SET(Can_FU.SteuReq[2],7); /*TIPP-*/
					FU.state_tipp_schnell = TRUE;
					FU.IdxIntern = 0;
				}
			}
			if (FU.state_tipp_minus && FU.cmd_tipp_schnell && !FU.state_tipp_schnell)
			{
				FU.IdxIntern ++;
				if(	FU.IdxIntern == WAITCYCLES)
				{
					if (MirroredMachine)
						Can_FU.SteuReq[2] = BIT_SET(Can_FU.SteuReq[2],7); /*TIPP-*/
					else
						Can_FU.SteuReq[2] = BIT_SET(Can_FU.SteuReq[2],6); /*TIPP-*/
					FU.state_tipp_schnell = TRUE;
					FU.IdxIntern = 0;
				}
			}

/* Kommando TIPP- oder + gegangen: einmal TIPP Bits rücksetzen */
			if (!FU.cmd_tipp_minus && !FU.cmd_tipp_plus)
			{
				Can_FU.SteuReq[2] = BIT_CLR(Can_FU.SteuReq[2],6); /*TIPP+*/
				Can_FU.SteuReq[2] = BIT_CLR(Can_FU.SteuReq[2],7); /*TIPP-*/
				FU.state_tipp_minus = 0;
				FU.state_tipp_plus = 0;
				FU.state_tipp_schnell = 0;
			}
		} /*else*/
	}

/********************************************************************/
/* Befehlsmerker senden*/
/********************************************************************/

	/* die Einzelmerker in das Steuerwort schreiben */
	Can_FU.SteuReq[3] = 0;
	j = 1;
	for(i=0;i<8;i++)
	{
		Can_FU.SteuReq[3] = Can_FU.SteuReq[3] | (j * FU.BefehlsMerker[i]);
		j *= 2;
	}

/*in jedem Zyklus das Schreibevent auslösen*/
	Can_FU.SteuReqEv = 1;

/********************************************************************/
/********************************************************************/
/********************************************************************/

/* Parameter SCHREIBEN Anforderung durch Applikation */
	if (FU.SetPara == 1)
	{
		switch (FU.ParaStep)
		{
			case 0:
			{
						/* Daten Eintragen */
				Can_FU.ParaReq[0] = FU_Param.ParaNr & 0x00FF;
				Can_FU.ParaReq[1] = (USINT)(FU_Param.ParaNr >> 8) & 0x00FF;
				/*FeldParameter -> andere Kennung und Index eintragen*/
				if(FU_Param.ParaNr == 728)
				{
					Can_FU.ParaReq[2] = FELD_PARAM_SEL;
					Can_FU.ParaReq[7] = FU_Param.Index;
				}
				/*StandardParameter */
				else
				{
					Can_FU.ParaReq[2] = STANDARD_PARAM_SEL;
					Can_FU.ParaReq[7] = 0;
				}
				tmpPtr = (UDINT*) &Can_FU.ParaReq[3];
				*tmpPtr = FU_Param.Wert;

				Can_FU.ParaReqEv = 1; 	/* Daten senden */
				FU.ParaStep = 1;
				FU_Param.Ready = 0;
				break;
			}
			case 1:
			{
			/*Rückmeldung vom FU erwarten und auswerten*/
				if(Can_FU.ParaResEv == 1)
				{
					Can_FU.ParaResEv = 0;
					/*Status OK?*/
					if (Can_FU.ParaRes[2] == 0)
					{
						FU.ParaStep = 2;
						FU_Param.Error = 0;
					}
					else
						FU_Param.Error = 1;
				}
				break;
			}
			case 2:
			{
				FU.SetPara = 0;
				FU.ParaStep = 0;
				FU_Param.Ready = 1;
			}
		} /*switch*/
	} /*if (FU.SetPara == 1)*/
}	/* Endcyclic */
```

- bit_func.h (reference to Logical/GlobalIncludes/bit_func.h)

- glob_var.h (reference to Logical/GlobalIncludes/glob_var.h)

#### lust_ref.c
```c
#ifdef _DEFAULT_INCLUDES
	#include <AsDefault.h>
#endif
/****************************************************************************/
/*	Referenzfahrt für LUST FU CDD3000 über CAN			 					*/
/*																			*/
/*																			*/
/*	Versionsgeschichte:														*/
/*  Version		Datum		Änderung								von		*/
/*	1.0			09.08.02	erste Implementation					HA		*/
/*																			*/
/*																			*/
/****************************************************************************/
#include "bit_func.h"				/*	Macros für die Bitbearbeitung		*/
#include "glob_var.h"
#include "math.h"

/****************************************************************************/
/*		DEFINES																*/
/****************************************************************************/
#define WAITCYCLES (200)

/****************************************************************************/
/*		Variablendeklaration												*/
/****************************************************************************/

/* Struktur für zu schreibende/lesende Parameter */
extern	FU_Para_Typ		FU_Param;
extern REAL ParkSpeed_Old;

_LOCAL USINT RefStep;
UINT WaitCounter;

void ReferenzFahrt(void)
{
/*V2.00 safety*/
	if(!FU.ENPO)
	{
		RefStep = 0;
		FU.cmd_Ref = 0;
		FU.BefehlsMerker[0] = FALSE;
	}
	if (!FU.cmd_Ref)
		RefStep = 0;

	switch (RefStep)
	{
		case 0:
		{
			if(FU.cmd_Ref)
				RefStep++;
			break;
		}
		case 1:
		{
		/* check, if no sending active*/
			if(!FU.SetPara)
			{
				RefStep++;
				FU_Param.Ready = FALSE;
			}
			break;
		}
		case 2:
		{
/* Wait for sending ready*/
			if(FU_Param.Ready)
			{
				FU_Param.Ready = FALSE;
				RefStep++;
			}
/* set data to send*/
			else
			{
				FU_Param.ParaNr = 724;
				FU_Param.Wert = (UDINT)(((float)X_Param.RefSpeed1) * X_Param.InkrementeProMm / 1000.0);
				FU.SetPara = 1;
			}
			break;
		}
		case 3:
		{
/* Wait for sending ready*/
			if(FU_Param.Ready)
			{
				FU_Param.Ready = FALSE;
				RefStep++;
			}
/* set data to send*/
			else
			{
				FU_Param.ParaNr = 725;
				FU_Param.Wert = (UDINT)(((float)X_Param.RefSpeed2) * X_Param.InkrementeProMm / 1000.0);
				FU.SetPara = 1;
			}
			break;
		}
		case 4:
		{
/* Wait for sending ready*/
			if(FU_Param.Ready)
			{
				FU_Param.Ready = FALSE;
				RefStep++;
			}
/* set data to send*/
			else
			{
				FU_Param.ParaNr = 726;
				FU_Param.Wert = (UDINT)(((float)X_Param.RefSpeed3) * X_Param.InkrementeProMm / 1000.0);
				FU.SetPara = 1;
			}
			break;
		}
		case 5:
		{
/* Wait for sending ready*/
			if(FU_Param.Ready)
			{
				FU_Param.Ready = FALSE;
				RefStep++;
			}
/* set data to send*/
			else
			{
		/* Parkposition */
				FU_Param.ParaNr = 728;
				FU_Param.Index = 14;
				FU_Param.Wert = (UDINT) (X_Param.ParkPosition * X_Param.InkrementeProMm);
				FU.SetPara = 1;
			}
			break;
		}
		case 6:
		{
/* Wait for sending ready*/
			if(FU_Param.Ready)
			{
				FU_Param.Ready = FALSE;
				RefStep++;
				ParkPositionChanged = 0;
				ParkSpeed_Old = X_Param.ParkSpeed;
			}
/* set data to send*/
			else
			{
		/* Parkspeed */
				FU_Param.ParaNr = 728;
				FU_Param.Index = 13;
				FU_Param.Wert = (UDINT)(((float)X_Param.ParkSpeed) * X_Param.InkrementeProMm / 1000.0);
				FU.SetPara = 1;
			}
			break;
		}
		case 7:
		{
			/* Wait for sending ready*/
						if(FU_Param.Ready)
						{
							FU_Param.Ready = FALSE;
							RefStep++;
						}
			/* set data to send*/
						else
						{
							FU_Param.Index = 0;
			/* manuell langsam */
							FU_Param.ParaNr = 716;
							FU_Param.Wert = (UDINT) (X_Param.ManSpeed1 * X_Param.InkrementeProMm / 1000.0);
							FU.SetPara = 1;
						}
						break;
		}
		case 8:
		{
			/* Wait for sending ready*/
						if(FU_Param.Ready)
						{
							FU_Param.Ready = FALSE;
							RefStep = 20;
						}
			/* set data to send*/
						else
						{
							FU_Param.Index = 0;
			/* manuell langsam */
							FU_Param.ParaNr = 715;
							FU_Param.Wert = (UDINT) (X_Param.ManSpeed2 * X_Param.InkrementeProMm / 1000.0);
							FU.SetPara = 1;
						}
						break;
		}

		case 9:
		{
/*Referenz triggern, wenn Rückmeldung nächster Schritt*/
			if(FU.BefehlsMerker[0] == TRUE && FU.ZustandsMerker[0] == TRUE)
			{
				RefStep++;
			}
			else
				FU.BefehlsMerker[0] = TRUE; /*Ref starten*/
			break;
		}
		case 10:
		{
/* auf Referenz fertig warten*/
			if(FU.ZustandsMerker[1])
			{
/*Befehl wegnehmen*/
				FU.BefehlsMerker[0] = FALSE; /**/
				RefStep++;
			}
			break;
		}
		case 11:
		{
/* auf weggehen der Rückmeldungen warten*/
			if( !FU.ZustandsMerker[0] && !FU.ZustandsMerker[0] )
			{
				RefStep++;
			}
			break;
		}
		case 12:
		{
			RefStep = 0;
			FU.cmd_Ref = 0;
			break;
		}

/*extra steps between 8 and 9 for starting auto mode*/
		case 20:
		{
			if(FU.Activ)
			{
				RefStep = 22;
				WaitCounter = 0;
				break;
			}
			FU.cmd_Start = 1;
			break;
		}
/*wait a little...*/
		case 22:
		{
			WaitCounter++;
			if(WaitCounter > WAITCYCLES)
			{
				WaitCounter = 0;
				RefStep = 25;
				break;
			}
			break;
		}

		case 25:
		{
			if(FU.Auto)
			{
				RefStep = 27;
				WaitCounter = 0;
				break;
			}
			FU.cmd_Auto = 1;
			break;
		}
/*wait a little...*/
		case 27:
		{
			WaitCounter++;
			if(WaitCounter > WAITCYCLES)
			{
				WaitCounter = 0;
				RefStep = 9;
				break;
			}
			break;
		}
	}
}
```

#### resetfudata.c
```c
#ifdef _DEFAULT_INCLUDES
	#include <AsDefault.h>
#endif
/****************************************************************************/
/*  	Hilfsfunktion														*/
/*		Rücksetzen der internen Statusinformation (State Machine)			*/
/****************************************************************************/

#include "bit_func.h"				/*	Macros für die Bitbearbeitung		*/
#include "glob_var.h"

/****************************************************************************/
/*		DEFINES																*/
/****************************************************************************/
extern CAN_OBJEKT_FUtyp	Can_FU;

/****************************************************************************/
/*		Rücksetzen der internen Statusinformation (State Machine)			*/
/****************************************************************************/
void resetFUData(void)
{
	int i;
/* Statusinformationen in Einzelbits intialisieren */
/* Byte 0 */
				FU.Error 			= FALSE;
				FU.CANStatus		= FALSE;
				FU.SollwertErreicht	= FALSE;
				FU.Activ 			= FALSE;
				FU.Rot0 			= FALSE;
				FU.CReady 			= FALSE;
/* Byte 1*/
				FU.ENPO 			= FALSE;
				FU.OSD00 			= FALSE;
				FU.OSD01 			= FALSE;
/* Byte 2 */
				FU.RefOk 			= FALSE;
				FU.Auto 			= FALSE;
				FU.Ablauf 			= FALSE;

				for (i=0;i<8;i++)
				{
					Can_FU.SteuReq[i] = 0;
					Can_FU.StatRes[i] = 0;
				}
}
```

#### lust_park.c
```c
#ifdef _DEFAULT_INCLUDES
	#include <AsDefault.h>
#endif
/****************************************************************************/
/*	Referenzfahrt für LUST FU CDD3000 über CAN			 					*/
/*																			*/
/*																			*/
/*	Versionsgeschichte:														*/
/*  Version		Datum		Änderung								von		*/
/*	1.0			09.08.02	erste Implementation					HA		*/
/*																			*/
/*																			*/
/****************************************************************************/
#include "bit_func.h"				/*	Macros für die Bitbearbeitung		*/
#include "glob_var.h"

/****************************************************************************/
/*		DEFINES																*/
/****************************************************************************/

/****************************************************************************/
/*		Variablendeklaration												*/
/****************************************************************************/

/* Struktur für zu schreibende/lesende Parameter */
extern	FU_Para_Typ		FU_Param;
extern REAL ParkSpeed_Old;

_LOCAL USINT ParkStep;

void ParkPosition(void)
{
/*safety!*/
	if(!FU.Activ || !FU.ENPO || !FU.Auto)
	{
		ParkStep = 0;
		FU.cmd_Park = 0;
		FU.BefehlsMerker[1] = FALSE;
		FU.BefehlsMerker[3] = FALSE;
	}
	if (!FU.cmd_Park)
		ParkStep = 0;

	switch (ParkStep)
	{
		case 0:
		{
			if(FU.cmd_Park)
			{
				if( (ParkPositionChanged)
				 || (abs(ParkSpeed_Old - X_Param.ParkSpeed)> 1)
				  )
					ParkStep++;
/* Parkpos unverändert: keine Parameterübergabe*/
				else
					ParkStep = 4;
			}
			break;
		}
		case 1:
		{
		/* check, if no sending active*/
			if(!FU.SetPara)
			{
				ParkStep++;
				FU_Param.Ready = FALSE;
			}
			break;
		}
		case 2:
		{
/* Wait for sending ready*/
			if(FU_Param.Ready)
			{
				FU_Param.Ready = FALSE;
				ParkStep++;
			}
/* set data to send*/
			else
			{
		/* Parkposition */
				FU_Param.ParaNr = 728;
				FU_Param.Index = 14;
				FU_Param.Wert = (UDINT) (X_Param.ParkPosition * X_Param.InkrementeProMm);
				FU.SetPara = 1;
			}
			break;
		}
		case 3:
		{
/* Wait for sending ready*/
			if(FU_Param.Ready)
			{
				FU_Param.Ready = FALSE;
				ParkStep++;
				ParkPositionChanged = 0;
				ParkSpeed_Old = X_Param.ParkSpeed;
			}
/* set data to send*/
			else
			{
		/* Parkspeed */
				FU_Param.ParaNr = 728;
				FU_Param.Index = 13;
				FU_Param.Wert = (UDINT)(((float)X_Param.ParkSpeed) * X_Param.InkrementeProMm / 1000.0);
				FU.SetPara = 1;
			}
			break;
		}
		case 4:
		{
/*Fahrt zur Parkpos triggern, wenn Rückmeldung nächster Schritt*/
			if(FU.BefehlsMerker[1] == TRUE && FU.ZustandsMerker[4] == TRUE)
			{
				ParkStep++;
			}
			else
				FU.BefehlsMerker[1] = TRUE; /* starten*/
			break;
		}
		case 5:
		{
/* auf fertig warten*/
			if(FU.ZustandsMerker[5])
			{
/*Befehl wegnehmen*/
				FU.BefehlsMerker[1] = FALSE; /**/
				ParkStep++;
			}
			break;
		}
		case 6:
		{
/* auf weggehen der Rückmeldungen warten*/
			if( !FU.ZustandsMerker[4] && !FU.ZustandsMerker[5] )
			{
				ParkStep++;
			}
			break;
		}
		case 7:
		{
			ParkStep = 0;
			FU.cmd_Park = 0;
			break;
		}
	}
}
```

#### lust_target.c
```c
#ifdef _DEFAULT_INCLUDES
	#include <AsDefault.h>
#endif
/****************************************************************************/
/*	Zielpos anfahren für LUST FU CDD3000 über CAN			 				*/
/*																			*/
/*																			*/
/*	Versionsgeschichte:														*/
/*  Version		Datum		Änderung								von		*/
/*	1.0			09.08.02	erste Implementation					HA		*/
/*																			*/
/*																			*/
/****************************************************************************/
#include "bit_func.h"				/*	Macros für die Bitbearbeitung		*/
#include "glob_var.h"

/****************************************************************************/
/*		DEFINES																*/
/****************************************************************************/

/****************************************************************************/
/*		Variablendeklaration												*/
/****************************************************************************/

/* Struktur für zu schreibende/lesende Parameter */
extern	FU_Para_Typ		FU_Param;
extern REAL ParkSpeed_Old;

_LOCAL USINT TargetStep;

void ZielPosition(void)
{

/*safety!*/
	if(!FU.Activ || !FU.ENPO || !FU.Auto)
	{
		TargetStep = 0;
		FU.cmd_Target = 0;
		FU.BefehlsMerker[1] = FALSE; /* starten*/
		FU.BefehlsMerker[3] = FALSE; /* starten*/
	}
	if (!FU.cmd_Target)
		TargetStep = 0;

	switch (TargetStep)
	{
		case 0:
		{
			if(!FU.cmd_Target)
				break;
		/* check, if no sending active*/
			if(!FU.SetPara)
			{
		/* Targetposition */
				FU_Param.ParaNr = 728;
				FU_Param.Index = 19;
				FU.TargetPosition = FU.TargetPosition_mm * X_Param.InkrementeProMm;
				FU_Param.Wert = FU.TargetPosition;
				FU.SetPara = 1;
				FU_Param.Ready = FALSE;
				TargetStep = 2;
			}
			break;
		}
		case 2:
		{
/* Wait for sending ready*/
			if(FU_Param.Ready)
			{
				FU_Param.Ready = FALSE;
				if (abs(ParkSpeed_Old - X_Param.ParkSpeed)< 1)
					TargetStep = 4;
				else
					TargetStep++;
			}
			break;
		}
		case 3:
		{
/* Wait for sending ready*/
			if(FU_Param.Ready)
			{
				FU_Param.Ready = FALSE;
				ParkSpeed_Old = X_Param.ParkSpeed;
				TargetStep++;
			}
/* set data to send*/
			else
			{
		/* Parkspeed */
				FU_Param.ParaNr = 728;
				FU_Param.Index = 13;
				FU_Param.Wert = (UDINT)(((float)X_Param.ParkSpeed) * X_Param.InkrementeProMm / 1000.0);
				FU.SetPara = 1;
			}
			break;
		}
		case 4:
		{
/*Fahrt zur Parkpos triggern, wenn Rückmeldung nächster Schritt*/
			if(FU.BefehlsMerker[3] == TRUE && FU.ZustandsMerker[4] == TRUE)
			{
				TargetStep++;
			}
			else
			{
				FU.BefehlsMerker[1] = TRUE; /* starten*/
				FU.BefehlsMerker[3] = TRUE; /* starten*/
			}
			break;
		}
		case 5:
		{
/* auf fertig warten*/
			if(FU.ZustandsMerker[5])
			{
/*Befehl wegnehmen*/
				FU.BefehlsMerker[1] = FALSE; /**/
				FU.BefehlsMerker[3] = FALSE; /**/
				TargetStep++;
			}
			break;
		}
		case 6:
		{
/* auf weggehen der Rückmeldungen warten*/
			if( !FU.ZustandsMerker[4] && !FU.ZustandsMerker[5] )
			{
				TargetStep = 0;
				FU.cmd_Target = 0;
			}
			break;
		}
	}
}
```

#### expose.c
```c
#ifdef _DEFAULT_INCLUDES
	#include <AsDefault.h>
#endif
/****************************************************************************/
/*	Belichtung für LUST FU CDD3000 über CAN				 					*/
/*																			*/
/*																			*/
/*	Versionsgeschichte:														*/
/*  Version		Datum		Änderung								von		*/
/*	1.0			14.08.02	erste Implementation					HA		*/
/*																			*/
/*																			*/
/****************************************************************************/
#include "bit_func.h"				/*	Macros für die Bitbearbeitung		*/
#include "glob_var.h"
#include "math.h"

/****************************************************************************/
/*		DEFINES																*/
/****************************************************************************/

/****************************************************************************/
/*		Variablendeklaration												*/
/****************************************************************************/

/* Struktur für zu schreibende/lesende Parameter */
extern	FU_Para_Typ		FU_Param;

_LOCAL USINT 	ExpStep;
REAL speed;
UDINT Vorkomma,Nachkomma;
/* Variablen f Altwerte*/
REAL 	speed_old,StartPosition_old,PEGStartPosition_old,EndPosition_old,
		PEGEndPosition_old;

void Belichtung(void)
{
/*safety!*/
	if(!FU.Activ || !FU.ENPO || !FU.Auto)
	{
		ExpStep = 0;
		FU.cmd_Expose = 0;
		FU.BefehlsMerker[2] = FALSE;
	}
	if (!FU.cmd_Expose)
		ExpStep = 0;

	switch (ExpStep)
	{
		case 0:
		{
			if(FU.cmd_Expose)
			{
		/*any Parameter changed? send all of them*/
				if( speed_old 				!= Expose_Param.ExposeSpeed 		||
					StartPosition_old 		!= Expose_Param.StartPosition 		||
					EndPosition_old 		!= Expose_Param.EndPosition 		||
					PEGStartPosition_old 	!= Expose_Param.PEGStartPosition 	||
					PEGEndPosition_old 		!= Expose_Param.PEGEndPosition 		)
					ExpStep++;
				else
			/* all parameters the same? jump to step 8 directly*/
					ExpStep = 8;
			}
			break;
		}
		case 1:
		{
		/* check, if no sending active*/
			if(!FU.SetPara)
			{
				ExpStep++;
				FU_Param.Ready = FALSE;
			}
			break;
		}
		case 2:
		{
/* Wait for sending ready*/
			if(FU_Param.Ready)
			{
				FU_Param.Ready = FALSE;
				StartPosition_old = Expose_Param.StartPosition;
				ExpStep++;
			}
/* set data to send*/
			else
			{
		/* Expose Start Position */
				FU_Param.ParaNr = 728;
				FU_Param.Index = 17;
				FU_Param.Wert = (UDINT) (Expose_Param.StartPosition * X_Param.InkrementeProMm);
				FU.SetPara = 1;
			}
			break;
		}
		case 3:
		{
/* Wait for sending ready*/
			if(FU_Param.Ready)
			{
				FU_Param.Ready = FALSE;
				PEGStartPosition_old = Expose_Param.PEGStartPosition;
				ExpStep++;
			}
/* set data to send*/
			else
			{
		/* PEG Start Position */
				FU_Param.ParaNr = 728;
				FU_Param.Index = 11;
				FU_Param.Wert = (UDINT) (Expose_Param.PEGStartPosition * X_Param.InkrementeProMm);
				FU.SetPara = 1;
			}
			break;
		}
		case 4:
		{
/* Wait for sending ready*/
			if(FU_Param.Ready)
			{
				FU_Param.Ready = FALSE;
				EndPosition_old = Expose_Param.EndPosition;
				ExpStep++;
			}
/* set data to send*/
			else
			{
		/* Expose End Position */
				FU_Param.ParaNr = 728;
				FU_Param.Index = 18;
				FU_Param.Wert = (UDINT) (Expose_Param.EndPosition * X_Param.InkrementeProMm);
				FU.SetPara = 1;
			}
			break;
		}
		case 5:
		{
/* Wait for sending ready*/
			if(FU_Param.Ready)
			{
				FU_Param.Ready = FALSE;
				PEGEndPosition_old = Expose_Param.PEGEndPosition;
				ExpStep++;
			}
/* set data to send*/
			else
			{
		/* PEG End Position */
				FU_Param.ParaNr = 728;
				FU_Param.Index = 12;
				FU_Param.Wert = (UDINT) (Expose_Param.PEGEndPosition * X_Param.InkrementeProMm);
				FU.SetPara = 1;
			}
			break;
		}
		case 6:
		{
/* Wait for sending ready*/
			if(FU_Param.Ready)
			{
				FU_Param.Ready = FALSE;
				ExpStep++;
			}
/* set data to send*/
			else
			{
		/* Expose speed Vorkomma Anteil*/
				FU_Param.ParaNr = 728;
				FU_Param.Index = 40;
				speed = Expose_Param.ExposeSpeed * X_Param.InkrementeProMm / 1000.0;
				Vorkomma = (UDINT) speed;
				Nachkomma = (UDINT)((speed - Vorkomma) * 10000.0);
				FU_Param.Wert = Vorkomma;
				FU.SetPara = 1;
			}
			break;
		}
		case 7:
		{
/* Wait for sending ready*/
			if(FU_Param.Ready)
			{
				FU_Param.Ready = FALSE;
				speed_old = Expose_Param.ExposeSpeed;
				ExpStep++;
			}
/* set data to send*/
			else
			{
		/* Expose speed Nachkomma Anteil*/
				FU_Param.ParaNr = 728;
				FU_Param.Index = 41;
				FU_Param.Wert = Nachkomma;
				FU.SetPara = 1;
			}
			break;
		}
		case 8:
		{
/*Belichten triggern, wenn Rückmeldung nächster Schritt*/
			if(FU.BefehlsMerker[2] == TRUE && FU.ZustandsMerker[2] == TRUE)
			{
				ExpStep++;
			}
			else
				FU.BefehlsMerker[2] = TRUE; /*Belichtung starten*/
			break;
		}
		case 9:
		{
/* auf Belichtung fertig warten*/
			if(FU.ZustandsMerker[3])
			{
/*Befehl wegnehmen*/
				FU.BefehlsMerker[2] = FALSE; /**/
				ExpStep++;
			}
			break;
		}
		case 10:
		{
/* auf weggehen der Rückmeldungen warten*/
			if( !FU.ZustandsMerker[2] && !FU.ZustandsMerker[3] )
			{
				ExpStep++;
			}
			break;
		}
		case 11:
		{
			ExpStep = 0;
			FU.cmd_Expose = 0;
			break;
		}
	}
}
```

### Program Logical/Exposer/Hardware/can_comm (ANSIC, version 1.00.0) - CAN Kommunikationstreiber

#### can_comm.c
```c
#ifdef _DEFAULT_INCLUDES
	#include <AsDefault.h>
#endif
/****************************************************************************/
/*	Kommunikationsroutine für CAN 						 					*/
/*																			*/
/*  - Öffnen der Schnittstelle im INIT Teil									*/
/*  - zyklisches bearbeiten der Tabellenorientierten Kommunikation			*/
/*																			*/
/*																			*/
/*	Versionsgeschichte:														*/
/*  Version		Datum		Änderung								von		*/
/*	1.0			06.08.02	erste Implemetation						HA		*/
/*																			*/
/****************************************************************************/

#include <bur/plctypes.h>
#include <can_lib.h>								/*prototypes of can_lib*/
#include <dataobj.h>								/*prototypes of dataobj*/

CANopen_typ _LOCAL CANopen_01;
CANdftab_typ _LOCAL CANdftab_01;
CANrwtab_typ _LOCAL CANrwtab_01;

/* === variables declaration === */
_LOCAL UDINT error_var;
_LOCAL USINT memorytype;
_LOCAL DatObjInfo_typ DOInfo;
_GLOBAL BOOL CAN_ok;

void _INIT init( void )								/*init part of task*/
{
	CANopen_01.enable = 1;
	CANopen_01.baud_rate = 25;						/*define baud rate - 250 kBit/s, 12 -> 125KB/s */
	CANopen_01.cob_anz = 20;							/*dfine number  of COB`s*/
/*	CANopen_01.device = (UDINT) "IF3"; */				/*define device*/
	CANopen_01.device = (UDINT) "SL1.SS1.IF1";
	CANopen_01.error_adr = (UDINT)&error_var;				/*define error adress*/
	CANopen(&CANopen_01);							/*initiate CANopen*/

	if( CANopen_01.status == 0)						/*check error level*/
	{
		DOInfo.enable = 1;
		DOInfo.pName = (UDINT) "can_tab";			/* Datenmodulname für CAN Objekte */

		/* Call FBK */
		DatObjInfo(&DOInfo);

		/* Verify status */
		if (DOInfo.status == 0)
		{
		 	CANdftab_01.enable = 1;
		 	CANdftab_01.us_ident = CANopen_01.us_ident;		/*set us_ident*/
		 	CANdftab_01.table_adr = DOInfo.pDatObjMem;			/*define adress of data module*/
			CANdftab_01.tab_num = DOInfo.len / 72;				/*define number of values*/
	 		CANdftab (&CANdftab_01);     				/*initiate CANdftab*/

			if(CANdftab_01.status == 0)						/*check error level*/
			{
				CANrwtab_01.enable = 1;
	 			CANrwtab_01.tab_ident=CANdftab_01.tab_ident;			/*set tab_id*/
				CAN_ok = 1;
			}
			else
				CAN_ok = 0;
		}/*if DOInfo.status==0*/
		else
			CAN_ok = 0;
	} /* if canopen01.status==0 */
	else
		CAN_ok = 0;
}

void _CYCLIC cyclic( void )							/*cyclic part of task*/
{
	if(CANdftab_01.status == 0)						/*check error level*/
	{
		CANrwtab(&CANrwtab_01); 					/*initiate CANwrtab*/
		CAN_ok = 1;

	}
	else
		CAN_ok = 0;

}
```

### Program Logical/Exposer/Hardware/in_out (ANSIC, version 1.00.0) - Variablen anlegen und Bearbeiten der E/As

#### in_out.c
```c
#ifdef _DEFAULT_INCLUDES
	#include <AsDefault.h>
#endif

#define _IN_OUT_C_SRC

#include "in_out.h"
#include "glob_var.h"
#include "egmglob_var.h"

_GLOBAL BOOL	BUSY;
_GLOBAL BOOL	ERROR,NEWERROR;
_GLOBAL BOOL	STANDBY;
_GLOBAL BOOL	Clock_1s;
/*HA 14.01.04 V1.71 implemented Stop pins on conveyor */
_GLOBAL	BOOL			StopPinsUp;
static TP_10ms_typ ConvLateralPulse;

_INIT void i(void)
{
/*safety! when machine is switched off, the grip closes
so we leave it closed at startup*/
	Out_PaperGripOn[LEFT] = ON;
	Out_PaperGripOn[RIGHT] = ON;
	ConvLateralPulse.IN = FALSE;

}

_CYCLIC void c(void)
{
	Module4[0] = Out_AdjustSuckerActive[1];
	Module4[1] = Out_AdjustSuckerActive[0];
	Module4[10] = Out_AdjustSignalCross;
	Module4[11] = Out_Horn;

	Module5[1] = Out_FeederHorActive;
	Module5[2] = Out_ConveyorbeltPinsUp;
	Module5[3] = Out_AdjustSuckerActive[2];
	Module5[4] = Out_CoverLockOn;

	if ( !PlateTransportSim )
	{
		Module4[2] = Out_FeederVacuumOn[0];
		Module4[3] = Out_FeederVacuumOn[1];
		Module4[4] = Out_FeederVacuumOn[2];
		Module4[5] = Out_FeederVacuumOn[3];
		Module4[6] = Out_AdjustSuckerVacuumOn[1];
		Module4[7] = Out_AdjustSuckerVacuumOn[0];
		Module4[8] = Out_AdjustSuckerVacuumOn[2];
		Module4[9] = Out_FeederVacuumOn[4];
	}
	else
	{
		Module4[2] = 0;
		Module4[3] = 0;
		Module4[4] = 0;
		Module4[5] = 0;
		Module4[6] = 0;
		Module4[7] = 0;
		Module4[8] = 0;
		Module4[9] = 0;
	}

	Module5[0] = !Out_PaperGripOn[LEFT]; /* both grippers via one output */
	Module5[5] = 0;
	Module5[6] = BUSY;
	Module5[7] = STANDBY;
	if (ERROR)
	{
		if (NEWERROR)
		{
			if (Clock_1s)
				Module5[8] = 1;
			else
				Module5[8] = 0;
		}
		else
			Module5[8] = 1;
	}
	else
		Module5[8] = 0;

	ConvLateralPulse.IN = Out_ConveyorbeltLateral;
	if( (DeloaderParameter.ConvLateralPulseTime > 0) && (DeloaderParameter.ConvLateralPulseTime < 500) )
		ConvLateralPulse.PT = DeloaderParameter.ConvLateralPulseTime;
	else
		ConvLateralPulse.PT = 50;

	TP_10ms(&ConvLateralPulse);

	Module5[9] = ConvLateralPulse.Q;
	Module5[10] = 0;
	Module5[11] = 0;

	Module6[0] = Out_AdjustPins4and6Up;
	Module6[1] = Out_AdjustPin3Up;
	Module6[2] = Out_AdjustPinsDown;
	Module6[3] = 0;
	Module6[4] = Out_LiftingPinsUp;
	Module6[5] = Out_LiftingPinsDown;
	if ( !PlateTransportSim )
	{
		Module6[6] = AdjustVacuumOn[0];
		Module6[7] = AdjustVacuumOn[1];
		Module6[8] = AdjustVacuumOn[2];
		Module6[9] = AdjustBlowairOn;
	}
	else
	{
		Module6[6] = 0;
		Module6[7] = 0;
		Module6[8] = 0;
		Module6[9] = 0;
	}
	Module6[10] = 0;
	Module6[11] = 0;

}
```

- in_out.h (reference to Logical/GlobalIncludes/in_out.h)

- glob_var.h (reference to Logical/GlobalIncludes/glob_var.h)

### Program Logical/Exposer/Hardware/seriell (ANSIC, version 1.10.0) - serielle Komm. mit Faulhaber Motoren
